(* IEC 61131-3 sources: advent-of-code/day9, 5 files *)

(* ---- demo.st ---- *)
VAR_GLOBAL CONSTANT
	rows : DINT := 5;
	cols : DINT := 10;
END_VAR

VAR_GLOBAL
	input : ARRAY[0..rows-1,0..cols -1] OF DINT :=
[
2,1,9,9,9,4,3,2,1,0,
3,9,8,7,8,9,4,9,2,1,
9,8,5,6,7,8,9,8,9,2,
8,7,6,7,8,9,6,7,8,9,
9,8,9,9,9,6,5,6,7,8
];
END_VAR

(* ---- input.st ---- *)
VAR_GLOBAL CONSTANT
	rows : DINT := 100;
	cols : DINT := 100;
END_VAR

VAR_GLOBAL
	input : ARRAY[0..rows-1,0..cols -1] OF DINT :=
[9,9,7,6,5,5,7,8,5,6,7,9,9,8,7,5,6,7,9,8,7,5,6,4,2,4,5,6,9,8,9,9,9,8,7,6,7,9,7,8,9,3,1,0,9,8,9,8,9,8,7,6,5,8,7,8,7,8,9,9,9,8,7,6,5,6,5,6,6,7,8,9,6,5,4,3,2,1,0,1,2,3,5,6,7,8,9,9,8,7,6,7,9,4,3,1,0,2,3,4,
8,7,6,5,4,3,2,1,4,5,7,8,9,9,8,3,9,8,9,8,6,4,3,2,1,3,4,5,9,7,8,9,9,9,9,5,4,5,6,9,5,3,2,9,8,7,6,7,9,9,6,5,4,2,6,5,6,7,8,9,9,8,6,5,4,2,3,4,5,7,8,9,9,6,5,4,3,2,9,4,3,9,6,9,8,9,8,7,6,6,5,6,7,9,4,4,2,5,4,5,
9,8,9,8,5,5,3,2,3,4,5,6,7,8,9,9,8,9,8,7,6,5,4,3,2,4,9,9,7,6,7,8,9,9,8,9,5,6,8,9,5,4,9,8,7,6,5,6,7,8,9,4,3,1,2,4,5,8,9,9,8,5,4,3,2,1,2,6,7,9,9,9,8,7,8,5,6,9,8,9,9,8,9,9,9,9,9,6,5,4,3,4,5,8,9,5,3,4,5,6,
8,9,8,7,6,6,8,7,6,5,6,7,9,9,9,8,7,6,9,9,8,6,7,5,3,9,8,7,6,5,6,7,9,8,7,9,9,8,9,9,6,9,8,7,6,5,4,5,6,7,8,9,1,0,1,3,4,5,6,9,7,6,5,4,3,2,3,5,6,7,8,9,9,8,9,6,7,9,7,9,8,7,8,9,9,9,8,9,5,4,2,5,5,7,8,9,4,5,9,7,
7,6,9,8,7,7,8,9,7,8,8,9,5,1,2,9,9,5,4,3,9,7,8,6,4,7,9,7,5,4,3,4,4,5,6,7,8,9,7,8,9,3,9,9,8,8,3,6,7,8,9,5,2,1,2,4,6,7,8,9,9,8,7,5,5,3,4,5,6,8,9,9,9,9,9,9,9,8,6,5,7,6,7,8,9,8,7,7,4,1,0,1,3,6,7,8,9,9,8,9,
7,5,3,9,9,8,9,9,8,9,9,4,3,2,3,9,8,6,5,2,9,8,9,8,5,6,9,8,4,3,2,1,3,4,7,9,9,6,5,4,3,2,9,8,7,6,2,3,8,9,5,4,3,2,4,5,8,8,9,2,1,9,7,6,6,4,6,8,9,9,8,8,9,9,9,8,7,6,5,4,3,5,6,9,8,7,6,5,3,2,1,2,4,5,6,9,5,6,7,8,
4,3,2,1,3,9,8,9,9,1,2,9,4,3,4,5,9,7,6,1,2,9,8,7,6,9,8,6,5,5,3,3,4,6,9,9,9,7,4,3,2,1,9,7,6,5,3,5,9,9,9,5,4,3,5,7,8,9,8,9,0,9,8,9,8,8,7,8,9,8,7,6,7,8,9,9,7,5,4,3,2,4,5,6,9,8,7,6,4,3,4,5,5,7,8,9,4,5,6,7,
9,9,3,2,3,5,7,8,9,0,9,8,9,4,9,6,9,8,7,2,3,5,9,9,9,8,9,8,7,6,4,4,5,7,8,9,8,7,5,2,1,0,2,9,7,6,9,9,8,7,8,9,7,5,6,8,9,9,7,8,9,9,9,9,9,9,9,9,7,6,5,5,6,6,8,9,8,6,5,5,4,6,8,9,4,9,8,7,6,7,8,9,6,7,9,4,2,4,5,6,
7,8,9,3,4,5,9,9,3,9,8,7,8,9,8,9,9,9,8,4,9,9,9,8,9,7,8,9,8,9,8,7,6,8,9,8,7,6,4,3,2,4,4,5,9,9,8,9,6,5,7,8,9,9,7,9,4,7,5,6,7,8,9,8,8,9,9,8,7,5,4,3,4,5,9,9,9,8,6,6,5,7,9,7,5,9,9,8,9,8,9,8,7,8,9,2,1,3,4,7,
6,8,9,9,9,7,8,9,1,9,9,6,5,5,7,8,9,9,9,9,8,7,8,7,5,6,7,8,9,9,9,9,7,8,9,9,8,7,5,4,3,9,5,6,9,9,7,8,9,4,6,8,9,9,8,9,3,3,4,5,8,9,8,7,7,9,8,6,5,4,3,2,3,6,7,8,9,9,8,7,6,8,9,7,6,8,9,9,2,9,3,9,8,9,8,4,2,5,6,8,
5,7,6,7,8,9,9,9,9,8,7,6,4,4,5,5,8,9,9,9,7,6,5,3,4,7,7,9,8,9,9,9,8,9,3,2,9,8,9,5,9,8,9,9,8,7,6,8,5,3,5,7,9,9,9,2,1,2,3,4,7,9,7,6,5,3,9,8,7,5,4,3,5,6,7,8,9,2,9,8,9,9,9,8,7,9,2,0,1,9,1,0,9,9,7,5,4,9,8,9,
4,3,5,6,8,9,9,9,8,7,6,4,3,2,3,4,7,8,9,9,8,7,4,1,3,5,6,6,7,8,9,9,9,8,9,1,2,9,8,9,8,7,9,9,8,7,5,3,1,2,3,8,9,9,4,3,0,1,6,5,6,9,8,7,6,4,5,9,8,9,5,9,6,7,8,9,4,3,4,9,2,1,0,9,8,9,3,9,9,8,9,1,9,8,7,6,9,8,9,9,
3,2,4,5,6,8,9,9,9,8,4,3,2,1,2,4,5,6,8,9,9,8,3,0,2,3,4,5,6,7,8,9,8,7,8,9,3,9,7,9,7,6,9,8,9,8,7,5,0,1,2,6,7,8,9,2,1,2,7,9,7,8,9,9,7,8,7,8,9,8,9,8,9,8,9,9,8,6,5,6,9,9,9,9,9,9,9,8,8,7,8,9,9,9,8,9,8,7,8,9,
4,3,4,6,8,9,7,9,9,8,5,4,3,3,4,5,6,8,9,8,6,3,2,1,2,5,5,8,7,8,9,7,9,6,9,9,9,8,6,8,7,5,7,7,8,9,9,4,2,3,3,4,5,9,9,4,3,3,4,5,8,9,9,8,9,9,9,9,8,7,7,7,8,9,9,9,9,7,6,9,8,7,8,9,9,9,8,7,6,5,7,8,9,9,9,8,7,6,4,5,
6,5,6,7,9,7,6,6,9,7,6,5,4,5,7,6,7,9,7,6,5,4,3,2,3,5,6,7,8,9,6,5,4,5,9,8,7,6,5,4,6,4,5,6,7,9,6,4,3,5,4,5,6,7,8,9,4,5,5,7,9,9,8,7,8,9,9,8,9,6,5,6,9,9,9,8,9,8,9,8,7,6,9,9,9,8,7,4,5,4,5,6,7,8,9,9,8,4,3,4,
7,9,8,8,9,6,5,4,9,8,8,6,5,6,8,7,8,9,9,8,7,5,4,3,4,5,7,8,9,8,7,8,5,6,9,9,8,7,6,3,2,3,8,9,9,8,7,5,9,8,5,6,7,8,9,7,5,7,8,9,9,8,7,6,7,9,8,7,6,5,3,7,8,9,8,7,8,9,8,7,6,5,6,8,9,9,6,3,2,3,4,5,6,7,8,9,4,3,2,3,
8,9,9,9,6,5,4,3,1,9,9,7,6,7,9,8,9,6,7,9,8,9,5,6,5,6,8,9,4,9,8,9,6,7,8,9,9,5,4,2,1,2,7,7,8,9,8,9,8,7,6,9,8,9,8,9,6,8,9,8,9,9,6,5,6,6,9,8,7,6,5,6,7,8,9,6,4,3,9,8,7,6,7,9,9,8,5,4,3,5,5,9,8,9,9,9,5,4,3,4,
9,4,9,8,7,6,5,4,2,3,4,9,8,8,9,9,6,5,6,7,9,8,7,7,9,8,9,4,3,2,9,8,7,8,9,9,8,7,4,3,2,3,5,6,7,8,9,9,9,8,8,9,9,6,7,8,9,9,8,7,7,6,5,4,5,5,4,9,8,7,6,7,8,9,8,9,3,2,1,9,9,7,8,9,8,7,6,9,8,6,6,7,9,8,7,8,9,6,4,5,
4,3,4,9,8,7,6,4,3,4,5,9,9,9,9,9,3,4,8,9,3,9,8,8,9,9,8,6,4,4,5,9,8,9,9,9,9,9,8,7,3,4,5,7,8,9,9,9,8,9,9,4,4,5,7,8,9,8,7,6,6,5,4,2,4,4,3,4,9,8,7,9,9,6,7,8,9,3,4,5,9,8,9,6,9,8,9,9,8,7,7,8,9,5,6,7,8,9,5,6,
3,2,5,6,9,8,7,5,9,5,9,8,9,8,8,8,9,9,9,4,2,3,9,9,4,3,9,9,5,7,8,9,9,7,8,7,9,9,9,6,5,6,8,9,9,8,9,8,7,6,5,3,2,1,6,7,8,9,6,5,4,3,2,1,0,1,2,3,4,9,8,9,6,5,7,9,9,4,9,7,8,9,3,4,5,9,9,9,9,8,9,9,2,4,5,6,9,9,6,9,
4,3,4,5,6,9,8,9,8,9,8,6,5,6,7,6,7,8,9,2,1,2,3,4,9,2,9,8,9,9,9,8,7,5,4,5,7,8,9,9,6,8,9,7,6,7,4,9,9,8,6,4,4,3,4,5,7,8,9,7,5,9,9,3,1,5,3,5,6,9,9,6,5,4,5,6,8,9,8,9,9,3,2,3,4,9,9,8,9,9,9,2,1,2,4,7,9,8,9,8,
9,5,5,9,8,9,9,8,7,6,5,4,3,1,3,4,6,9,4,3,2,5,4,9,8,9,8,7,8,9,9,7,6,4,3,4,5,6,9,8,7,9,7,6,5,4,3,9,8,7,6,5,6,7,5,6,7,8,9,9,9,7,8,9,2,3,4,6,9,8,5,4,3,2,3,4,5,6,7,8,9,4,3,9,9,8,7,7,7,8,7,9,9,3,9,9,8,7,8,7,
7,9,9,8,9,4,2,9,6,5,4,2,1,0,1,2,3,4,9,4,3,4,9,9,7,8,7,6,7,9,8,6,2,1,2,3,4,8,9,9,9,9,9,8,6,5,2,3,9,9,7,7,7,8,8,7,8,9,9,8,7,6,9,8,9,4,6,9,8,7,6,5,2,1,2,6,9,8,9,9,7,5,9,8,9,5,6,6,5,4,6,8,8,9,8,7,6,5,4,6,
6,8,9,7,8,9,1,9,7,7,6,3,2,1,6,3,7,6,8,9,4,9,8,7,6,5,6,5,6,8,9,5,4,0,1,3,5,6,7,9,9,9,8,7,5,2,1,4,5,6,9,8,8,9,9,8,9,8,7,7,6,5,8,7,7,9,9,9,9,8,7,6,3,2,3,4,9,9,1,0,9,9,8,7,7,4,5,2,3,3,5,6,7,9,9,8,5,4,3,4,
5,9,5,6,7,8,9,8,7,6,5,4,3,2,4,5,6,8,9,7,6,9,9,5,4,4,3,4,5,7,8,9,3,2,3,4,8,7,9,9,9,8,9,5,4,3,2,3,4,9,9,9,9,5,4,9,8,7,6,5,4,4,6,5,6,8,8,9,9,9,9,5,4,7,5,6,7,8,9,1,9,8,7,6,5,3,2,1,0,2,5,8,9,9,9,7,4,3,2,3,
3,3,4,7,9,7,9,9,9,7,6,5,9,4,5,6,7,8,9,8,9,8,7,4,3,1,2,5,5,6,7,8,9,6,5,5,6,9,9,9,8,7,8,9,5,6,3,9,9,8,7,6,7,4,3,4,9,8,9,4,3,3,3,4,5,6,7,8,9,9,9,7,5,6,7,8,9,9,8,9,8,9,8,7,6,4,3,2,1,3,4,6,7,9,7,6,5,4,3,4,
1,2,3,4,5,6,7,9,9,8,7,6,7,7,6,8,9,9,9,9,8,7,6,5,9,0,1,2,3,8,9,9,8,7,6,6,9,8,9,8,7,6,7,8,9,8,9,8,9,9,5,4,3,4,2,3,4,9,8,3,2,1,2,3,4,7,9,9,9,9,8,7,6,9,8,9,5,4,6,9,7,6,9,8,7,5,6,3,2,4,5,6,7,8,9,7,6,7,5,5,
3,5,6,9,6,7,8,9,6,9,8,8,9,8,7,9,8,9,8,9,9,8,7,9,8,9,2,3,5,6,8,9,9,8,7,9,8,7,8,9,6,5,9,9,9,9,9,6,9,8,9,5,2,0,1,2,9,8,7,5,3,3,3,4,5,6,7,8,9,1,9,8,7,8,9,5,4,3,9,7,6,5,9,8,7,6,7,5,6,5,6,7,8,9,9,8,8,7,6,7,
4,6,7,8,9,8,9,6,5,7,9,9,6,9,9,8,7,8,7,8,9,9,9,8,7,8,9,4,5,6,7,9,9,9,9,7,9,6,7,8,9,4,5,8,9,9,7,5,6,7,8,9,2,1,2,4,5,9,8,9,6,5,6,7,9,7,8,9,5,3,9,9,8,9,9,8,5,9,8,6,5,4,3,9,9,8,9,9,7,7,7,8,9,3,2,9,9,8,7,8,
6,9,8,9,2,9,8,7,4,3,2,3,5,9,8,7,6,5,6,7,9,9,9,8,6,7,8,9,7,8,9,3,9,8,7,6,8,5,9,9,4,3,4,6,9,8,6,4,5,6,9,8,9,2,4,5,9,9,9,8,7,7,9,8,9,8,9,7,6,9,8,6,9,8,9,7,6,9,8,7,6,5,4,7,8,9,6,7,9,8,9,9,6,5,4,5,9,9,8,9,
7,8,9,2,0,1,9,6,5,1,0,1,9,8,7,6,5,4,5,8,9,9,8,7,5,6,7,8,9,9,0,2,3,9,8,4,3,4,8,9,3,2,1,9,8,6,5,3,4,5,6,7,8,9,5,9,8,9,9,9,8,9,3,9,5,9,9,8,9,8,7,5,6,7,8,9,9,9,9,8,9,6,5,6,9,5,4,6,5,9,9,9,9,6,5,9,8,7,9,6,
8,9,8,9,1,9,8,7,7,2,1,2,4,9,8,5,4,3,4,5,9,9,9,8,9,8,8,9,7,8,9,3,4,9,6,5,2,5,7,8,9,9,9,8,9,8,4,2,3,4,9,8,9,9,9,8,7,8,9,8,9,0,1,2,3,9,9,9,9,9,6,4,6,7,9,6,8,9,9,9,9,7,6,7,8,9,3,3,4,9,8,9,8,9,6,9,7,6,5,4,
9,6,7,8,9,4,9,9,8,9,2,3,4,9,9,7,5,2,3,6,7,8,9,9,2,9,9,7,6,7,8,9,9,8,5,4,3,4,5,6,7,8,9,7,8,9,2,1,2,3,4,9,8,9,8,9,5,6,5,7,8,9,9,3,9,8,9,8,9,8,7,3,1,2,3,4,6,7,9,9,9,8,9,8,9,3,2,1,9,8,7,6,7,9,7,9,8,7,9,3,
3,5,6,8,9,3,1,0,9,8,9,4,9,8,8,6,2,1,2,7,8,9,7,5,1,0,3,4,5,6,7,9,8,7,6,5,4,5,6,7,8,9,8,6,9,8,9,0,1,2,9,8,7,9,7,5,4,3,4,9,9,9,8,9,8,7,6,7,8,9,8,2,0,1,2,4,5,6,7,8,9,9,9,9,9,9,1,0,1,9,9,5,6,8,9,9,9,9,8,9,
8,6,8,9,5,4,3,9,8,7,8,9,8,7,7,5,1,0,2,4,5,7,9,4,2,1,2,3,4,5,7,9,9,8,8,6,5,6,8,9,9,6,5,4,5,7,9,9,2,9,9,9,6,9,7,6,2,1,9,8,9,8,7,5,4,6,5,6,9,8,9,3,1,4,3,5,7,8,9,9,6,7,9,8,9,8,9,1,3,9,8,4,5,9,9,9,9,8,7,6,
8,7,9,7,6,9,9,8,7,6,9,8,7,6,5,4,3,2,3,5,6,8,9,4,3,2,3,4,5,6,7,9,8,9,9,7,6,7,9,9,9,5,4,3,5,4,9,8,9,8,7,6,5,4,3,2,1,0,1,7,8,9,5,4,3,2,4,9,8,7,8,9,2,3,8,7,9,9,1,3,4,9,8,7,7,6,8,9,9,8,7,3,7,8,9,8,9,7,6,5,
9,8,9,8,9,8,7,6,5,4,5,9,9,8,7,5,4,6,4,8,9,9,7,5,4,3,4,5,7,8,9,8,7,6,9,8,8,8,9,8,8,9,0,1,2,3,9,7,6,9,9,8,6,7,9,6,3,3,2,6,7,8,9,3,2,1,9,8,7,6,7,8,9,9,9,8,9,1,0,5,9,8,7,6,5,5,7,8,9,9,6,5,6,9,8,7,6,5,4,3,
3,9,7,9,9,9,8,9,4,3,4,5,6,9,8,7,5,9,6,7,8,9,9,6,5,9,5,6,8,9,9,9,6,5,4,9,9,9,9,7,6,8,9,3,5,9,8,9,5,6,7,9,7,9,8,5,4,5,4,5,6,7,8,9,4,3,9,7,6,5,6,7,6,7,8,9,3,2,1,6,7,9,6,5,4,3,5,6,9,8,7,6,7,9,9,8,7,6,5,4,
4,5,6,8,9,8,9,8,9,4,5,6,9,9,9,8,6,8,7,8,9,2,9,7,9,8,7,7,9,1,9,8,9,4,3,4,5,9,8,6,4,7,8,9,9,8,6,5,4,5,6,7,9,8,7,6,5,6,5,6,7,9,9,6,5,9,8,7,5,4,3,5,5,6,9,8,9,4,5,9,9,8,5,4,3,2,4,5,6,9,9,7,8,9,9,9,9,7,6,5,
5,6,9,9,8,7,6,7,9,5,6,7,8,9,6,9,7,8,8,9,2,1,9,8,9,9,8,9,1,0,9,7,8,9,4,9,9,8,9,4,3,5,1,9,8,9,7,4,3,4,5,6,7,9,8,7,6,7,6,7,8,9,8,7,9,8,7,6,4,3,2,3,4,5,6,7,8,9,9,8,7,6,5,4,2,1,2,3,4,7,9,8,9,9,9,8,7,9,7,6,
6,9,8,9,9,6,5,6,8,9,7,8,9,4,5,9,8,9,9,5,4,2,4,9,8,9,9,9,9,9,8,6,7,8,9,8,7,6,4,3,2,1,0,5,7,8,9,3,2,3,4,5,6,7,9,8,7,8,7,8,9,8,9,8,9,9,8,7,9,2,1,2,3,6,7,6,8,9,9,9,6,5,4,3,2,0,1,4,5,6,7,9,2,9,8,7,6,9,8,7,
9,9,7,6,8,6,4,5,7,8,9,9,4,3,4,4,9,8,9,6,5,6,9,8,7,9,9,9,8,7,6,5,3,4,9,8,7,6,5,4,5,9,2,4,6,9,3,2,1,2,3,6,7,8,9,9,8,9,8,9,9,7,8,9,3,2,9,9,8,9,0,1,2,3,4,5,7,8,9,9,8,7,8,4,3,1,2,3,4,5,8,9,1,2,9,6,5,6,9,8,
8,9,8,5,9,2,3,4,6,7,8,9,0,1,2,3,4,7,8,9,6,8,9,7,6,8,9,9,9,8,7,6,2,1,2,9,8,7,6,6,7,8,4,5,7,8,9,1,0,1,2,3,4,9,9,9,9,3,9,9,8,5,4,3,2,1,9,8,7,9,1,9,3,4,5,6,8,9,1,2,9,8,9,5,4,4,3,4,5,6,8,9,2,9,8,9,4,5,6,9,
7,6,5,4,3,1,2,3,5,6,9,2,1,3,5,4,5,6,7,8,9,9,8,6,5,6,7,8,9,9,8,5,4,2,3,7,9,8,7,9,8,9,7,6,9,9,3,2,1,2,3,4,5,6,8,9,3,2,9,8,7,6,5,4,5,9,8,7,6,8,9,8,9,5,6,9,9,1,0,1,2,9,8,6,5,6,7,7,6,7,9,9,9,8,6,4,3,4,5,9,
7,8,4,2,1,0,1,2,3,9,8,9,2,4,6,5,6,7,9,9,9,9,6,5,4,5,6,7,9,9,9,6,5,3,4,5,7,9,8,9,9,8,9,7,8,9,4,3,2,5,4,5,6,9,9,6,5,3,9,9,8,7,6,7,6,9,7,6,5,7,9,7,8,9,7,8,9,2,3,4,5,7,9,7,8,7,8,8,9,8,9,9,9,8,7,6,4,5,7,8,
6,5,4,3,2,1,4,3,5,6,7,8,9,5,6,8,7,9,9,9,9,8,7,3,2,3,5,6,8,9,9,7,6,4,5,6,8,9,9,7,6,7,9,8,9,6,5,4,3,7,5,6,7,8,9,9,7,9,8,9,9,8,7,9,8,9,8,7,4,4,5,6,7,8,9,9,9,4,4,7,6,7,9,8,9,8,9,9,8,9,9,8,9,9,8,6,5,7,8,9,
7,6,5,4,5,2,5,4,8,7,8,9,7,6,8,9,8,9,9,8,7,6,4,2,0,1,2,4,6,7,8,9,7,5,7,8,9,9,9,6,4,3,1,9,9,7,6,7,9,8,9,8,8,9,8,9,9,8,7,9,9,9,8,9,9,9,9,9,3,2,9,7,8,9,6,7,8,9,9,9,8,8,9,9,9,9,8,7,6,7,8,7,8,9,9,7,7,8,9,7,
8,7,7,5,6,8,6,5,9,8,9,7,9,7,9,9,9,9,8,7,6,5,4,3,1,2,8,5,7,8,9,9,9,6,7,9,9,9,8,7,5,4,9,9,8,9,9,8,9,9,8,9,9,5,7,8,9,9,6,7,8,9,9,4,5,9,8,7,6,3,7,9,9,5,4,5,9,8,8,9,9,9,1,2,9,8,7,6,5,6,7,6,9,8,9,9,8,9,5,6,
9,9,8,9,8,8,7,6,7,9,8,6,5,9,8,8,9,9,9,8,9,6,5,4,2,3,7,6,7,9,8,9,8,7,8,9,9,9,9,9,6,9,8,7,7,7,8,9,9,9,7,6,5,4,6,7,8,9,5,6,9,9,6,5,6,9,9,8,5,4,6,7,8,9,3,4,5,6,7,8,9,8,9,9,9,8,6,5,4,6,6,5,6,7,8,9,9,3,4,9,
5,6,9,8,9,9,8,9,8,9,5,3,4,5,6,7,9,9,8,9,8,7,6,6,4,5,6,7,9,8,7,6,9,9,9,8,8,9,3,1,9,8,7,6,5,6,7,8,9,9,8,8,7,2,3,4,9,9,4,3,9,8,7,6,9,8,9,9,6,5,7,9,9,1,2,3,6,9,8,9,8,7,6,8,9,6,5,4,3,1,5,4,5,6,7,9,1,2,9,8,
4,5,6,7,8,9,9,9,9,8,6,7,6,9,7,9,8,8,7,6,9,9,7,7,5,6,7,9,9,9,9,5,3,2,1,6,7,8,9,9,8,9,4,3,4,5,6,7,8,9,9,9,8,3,4,5,6,8,9,2,1,9,8,9,8,7,9,8,7,6,8,9,3,2,4,4,5,6,9,7,5,4,5,9,8,7,6,5,4,0,2,3,6,7,8,9,3,9,8,7,
5,9,8,9,9,8,9,7,6,9,9,8,9,8,9,7,6,5,4,5,4,5,9,8,6,7,9,9,8,9,8,9,5,4,3,5,8,9,9,8,7,6,5,4,5,6,7,8,9,3,2,1,9,4,6,7,8,9,9,1,0,1,9,8,7,6,5,9,8,7,8,9,4,9,9,7,6,8,9,6,4,3,4,5,9,8,9,7,5,1,4,5,8,9,9,9,9,9,9,6,
6,7,9,5,6,7,8,9,9,9,9,9,8,7,9,6,5,4,3,2,3,5,6,9,7,9,9,8,7,6,7,8,9,5,4,6,9,9,9,9,8,7,6,5,6,7,8,9,8,9,4,3,4,9,7,8,9,9,8,9,1,9,8,7,6,5,4,5,9,8,9,9,9,8,8,9,7,8,9,6,5,2,6,6,7,9,5,9,7,7,6,6,8,9,8,9,8,9,8,7,
7,8,9,4,5,6,9,8,7,8,9,9,7,6,8,9,6,3,2,1,2,3,9,9,8,9,8,9,6,5,6,9,7,6,9,7,9,9,8,1,9,8,7,6,9,8,9,6,7,9,6,4,5,9,8,9,9,8,7,8,9,9,9,9,7,4,3,4,5,9,9,8,7,6,7,9,9,9,7,5,4,3,4,8,9,5,4,2,9,8,7,8,9,6,7,9,7,6,9,9,
8,9,3,2,3,9,8,7,6,7,5,8,6,5,7,9,7,4,3,4,3,4,8,9,9,9,7,8,9,4,5,8,9,7,8,9,8,8,7,0,1,9,8,7,9,9,4,5,9,8,9,5,7,9,9,8,7,8,6,8,9,9,9,8,4,3,2,3,6,9,8,7,6,5,6,8,8,9,8,7,6,4,6,7,8,9,3,1,0,9,9,9,4,5,6,8,9,4,3,1,
9,5,4,3,9,8,7,6,5,6,3,2,3,4,8,9,8,5,4,5,7,5,6,9,8,6,5,6,9,3,4,7,8,9,9,8,7,6,5,3,2,3,9,9,1,2,3,4,9,7,8,9,9,8,7,9,6,4,5,6,7,8,9,6,5,4,3,4,9,8,9,6,7,4,5,6,7,8,9,8,9,8,7,9,9,9,9,2,9,9,8,7,5,6,7,9,7,2,1,0,
8,6,6,5,7,9,6,5,4,6,2,1,2,3,4,9,9,6,5,6,8,9,9,8,7,5,4,5,8,9,5,6,7,8,9,9,9,7,9,5,3,5,6,7,9,9,4,9,8,6,7,8,9,8,6,5,4,3,4,5,6,9,8,9,6,5,4,9,8,7,6,5,2,3,4,5,8,9,1,9,4,9,8,9,8,7,8,9,8,9,9,8,9,8,9,6,5,4,2,3,
9,9,7,6,9,8,7,6,3,2,1,0,1,4,6,7,8,9,6,7,9,8,5,5,4,4,3,6,7,8,9,7,8,9,4,3,9,8,9,6,9,8,7,8,9,8,9,8,7,5,6,7,9,6,5,4,3,2,3,4,5,6,7,8,9,6,9,8,8,7,4,3,1,3,3,7,9,9,0,1,3,4,9,8,7,6,7,8,7,8,9,9,6,9,8,7,6,6,7,5,
5,6,9,8,9,9,9,5,4,3,2,3,2,3,4,5,6,9,7,9,8,7,4,3,2,1,2,4,5,9,2,9,9,5,4,2,3,9,9,7,9,9,9,9,6,7,8,9,6,4,5,9,8,7,6,5,2,1,2,5,6,8,9,9,9,9,8,7,7,6,2,1,0,1,2,6,7,8,9,9,9,9,8,7,6,5,9,8,6,8,9,7,5,6,9,8,9,7,7,6,
3,5,6,9,8,9,8,6,7,4,3,4,6,5,5,6,7,8,9,9,9,6,5,4,9,0,3,6,6,9,3,9,8,7,5,4,9,9,7,9,3,2,3,4,5,6,7,8,9,3,4,5,9,8,7,4,3,2,7,6,8,9,9,9,9,8,7,6,5,4,3,2,1,2,3,4,5,9,8,7,8,9,9,8,9,4,3,4,5,6,8,9,3,4,5,9,5,9,8,7,
8,6,9,8,7,9,8,7,6,5,4,5,6,6,8,7,8,9,9,9,8,9,6,9,8,9,4,5,7,8,9,9,9,9,7,9,8,7,6,5,4,4,4,5,7,8,9,9,3,2,3,4,8,9,6,5,4,5,6,7,9,9,8,8,7,9,8,7,6,5,4,3,8,7,5,6,7,8,9,5,7,8,9,9,8,6,2,3,4,5,7,8,9,9,6,9,4,5,9,8,
9,9,8,7,6,5,9,8,7,8,7,6,7,7,9,8,9,9,9,8,7,8,9,8,7,9,5,7,8,9,7,8,8,9,9,9,9,8,7,9,5,5,6,9,8,9,6,5,4,3,4,6,7,9,8,9,5,9,8,9,9,9,7,6,5,4,9,8,8,7,6,5,9,8,6,7,8,9,5,4,8,9,8,7,6,5,3,4,6,6,9,9,9,8,9,8,9,9,9,9,
5,6,9,9,8,4,5,9,8,9,9,7,9,8,9,9,2,9,8,7,6,7,8,9,6,8,9,8,9,8,6,5,7,8,9,9,8,9,8,9,6,6,9,9,9,8,7,6,5,4,5,7,8,9,9,7,6,7,9,9,9,8,9,5,3,2,6,9,9,8,7,6,7,9,9,8,9,6,5,3,4,5,9,9,7,6,4,5,9,7,8,9,8,7,7,6,7,8,9,9,
4,9,8,7,6,3,1,2,9,6,9,8,9,9,3,2,1,0,9,6,5,6,3,5,5,7,8,9,9,7,5,4,6,7,9,8,7,8,9,8,7,9,8,8,8,9,9,7,6,7,6,9,9,7,9,9,7,8,9,9,8,7,8,9,4,3,5,6,7,9,8,7,8,9,9,9,8,7,9,4,6,9,9,9,8,7,5,6,7,8,9,8,9,6,6,4,6,7,8,9,
3,9,8,6,5,4,2,3,4,5,6,9,8,6,5,4,9,9,8,7,4,3,2,3,4,6,7,8,9,5,4,3,8,9,8,7,6,5,6,9,8,9,7,6,7,9,8,9,9,8,7,8,9,6,7,9,8,9,8,7,7,6,9,8,9,4,5,7,9,7,9,8,9,9,9,9,9,9,8,9,9,8,9,9,9,8,6,7,8,9,8,7,6,5,4,3,4,8,9,0,
4,9,8,7,6,5,3,4,5,7,7,8,9,7,9,9,7,7,5,8,1,0,1,2,4,5,8,9,6,4,3,2,9,8,7,6,5,4,5,6,9,8,6,5,6,5,6,7,8,9,8,9,5,5,6,2,9,9,9,5,6,5,6,7,8,9,6,8,9,6,5,9,9,8,7,8,9,8,7,8,8,7,8,9,9,9,9,8,9,2,9,8,5,4,3,2,4,6,9,1,
5,6,9,8,7,6,7,8,7,8,8,9,2,9,8,7,6,5,4,3,2,1,2,3,8,8,9,9,9,5,5,1,2,9,8,9,2,3,4,9,8,7,6,4,6,4,8,9,9,9,9,5,4,3,2,1,9,8,8,4,3,4,7,7,8,9,7,9,9,9,3,2,3,4,5,9,7,6,5,6,7,6,9,9,8,7,9,9,0,1,3,9,9,2,0,1,3,9,8,9,
9,9,7,9,8,7,8,9,8,9,9,9,1,0,9,8,7,7,5,5,4,3,6,4,6,7,8,9,8,7,6,3,9,9,9,8,9,4,9,8,7,6,5,3,4,3,4,8,7,8,9,6,5,4,6,2,9,7,6,5,2,3,4,6,9,6,9,7,8,8,9,1,2,3,9,9,8,3,4,3,4,5,8,9,9,6,9,5,3,2,4,9,8,9,3,2,9,9,7,8,
8,7,6,7,9,8,9,7,9,6,7,8,9,9,8,9,9,8,7,6,5,5,7,5,7,8,9,9,9,8,7,9,8,8,6,7,8,9,9,7,6,5,4,2,1,2,3,4,6,7,9,7,7,5,7,9,8,6,5,4,3,4,5,7,9,5,6,5,6,7,8,9,3,9,8,7,3,2,1,2,5,6,7,8,9,5,8,9,4,3,9,8,7,8,9,9,8,9,6,7,
7,6,5,6,8,9,6,5,4,5,6,7,8,9,7,6,5,9,8,8,6,6,8,6,9,9,9,8,9,9,9,8,7,6,5,1,2,9,8,7,6,5,4,3,0,1,2,3,7,8,9,8,8,6,8,9,9,7,6,5,4,5,7,9,5,4,4,4,5,6,7,8,9,8,7,5,4,5,2,3,8,7,8,9,3,4,7,8,9,9,8,7,6,7,9,8,7,6,5,6,
9,7,3,8,9,9,8,4,3,7,8,9,9,8,6,5,3,2,9,8,7,7,9,7,8,9,5,6,7,9,8,7,6,5,4,3,3,4,9,6,5,4,3,2,1,2,5,7,8,9,9,9,9,7,8,9,9,8,7,8,5,9,8,9,4,3,2,3,4,5,6,7,8,9,8,6,5,6,3,5,9,8,9,5,4,5,6,7,9,6,9,6,5,9,8,7,6,5,4,4,
7,6,2,9,6,8,9,5,4,5,6,7,8,9,7,4,3,1,0,9,8,9,9,8,9,4,3,2,3,4,9,9,8,6,5,9,5,9,8,7,8,5,4,3,2,3,4,5,6,8,9,3,9,8,9,1,2,9,8,9,6,7,9,2,1,0,1,5,6,7,8,9,9,9,9,7,6,5,4,5,6,9,7,6,7,6,7,9,8,5,4,5,4,6,9,8,5,4,3,3,
5,4,3,4,5,7,8,9,5,9,8,9,9,7,6,5,4,5,1,3,9,8,9,9,6,5,4,5,6,8,9,5,9,7,6,8,9,8,9,8,9,6,5,4,5,4,5,7,8,9,1,2,4,9,4,2,9,8,9,8,7,8,9,3,2,4,3,4,5,9,9,9,8,9,9,9,8,6,7,6,8,9,9,7,8,8,9,8,7,6,3,4,3,4,5,9,9,2,1,2,
6,5,4,5,7,8,9,7,6,7,9,5,3,9,8,6,5,3,2,5,6,7,9,8,7,8,5,6,7,8,9,4,9,8,7,9,8,7,6,9,9,7,6,5,7,9,7,8,9,8,9,4,9,9,9,9,8,7,9,9,8,9,5,4,9,5,6,5,9,8,7,8,7,8,9,5,9,7,9,7,9,9,9,8,9,9,8,7,6,6,2,1,2,5,9,8,8,3,0,1,
7,8,5,6,8,9,2,9,7,9,8,9,2,3,9,7,6,4,5,6,9,8,9,9,8,9,6,9,8,9,2,3,5,9,9,8,9,6,5,6,7,9,7,6,7,9,8,9,6,7,9,9,8,9,8,9,7,6,5,6,9,8,7,9,8,9,7,9,8,7,6,7,6,7,9,6,9,8,9,9,9,9,6,9,9,8,7,6,5,4,3,0,1,9,8,7,6,3,1,2,
8,7,6,9,9,2,1,9,8,9,7,9,9,4,9,8,7,7,6,7,8,9,5,6,9,8,7,8,9,9,9,4,5,9,8,7,6,5,4,5,7,9,8,7,8,9,9,4,5,6,9,8,7,8,7,8,9,5,4,5,6,9,9,9,7,6,9,8,7,6,5,8,5,6,8,9,9,9,9,9,9,8,5,6,7,9,8,7,6,5,3,2,3,6,9,9,5,4,2,3,
9,8,7,8,9,3,2,9,9,8,6,8,8,9,9,9,9,8,7,8,9,3,4,9,9,9,8,9,6,9,8,9,9,8,7,6,5,4,3,4,9,8,9,8,9,0,1,9,9,9,8,7,6,5,6,9,6,5,3,4,5,9,8,7,6,5,6,9,8,7,4,3,4,5,6,7,8,9,9,8,7,6,4,3,9,7,9,8,7,6,5,3,4,5,9,8,6,5,6,4,
8,9,8,9,5,4,9,8,7,6,5,6,7,8,9,6,8,9,8,9,9,2,9,8,9,7,9,6,5,8,7,8,9,9,9,8,7,3,2,5,6,7,9,9,3,1,9,8,7,6,5,4,5,4,5,8,9,3,2,3,9,8,7,6,5,4,5,9,8,7,3,2,3,4,8,9,9,1,0,9,8,7,6,4,9,6,4,9,9,7,6,4,5,6,7,9,8,7,7,5,
7,4,9,7,6,5,7,9,8,8,4,5,6,9,5,4,5,5,9,7,8,9,8,7,6,5,7,2,4,5,6,7,9,9,8,7,5,4,5,6,7,8,9,8,9,9,9,9,6,5,4,3,2,3,6,7,8,9,1,2,9,7,6,6,4,3,4,5,9,6,5,4,4,5,9,5,4,3,9,9,9,8,7,9,8,4,3,2,9,8,9,9,8,7,8,9,9,8,8,9,
6,5,6,9,8,7,8,9,9,9,5,6,7,8,9,3,2,4,5,6,9,9,7,9,8,3,4,1,2,4,8,6,7,8,9,9,9,5,7,8,9,9,8,6,5,8,7,8,9,6,5,4,1,2,7,6,7,9,2,9,7,6,5,4,3,2,3,9,8,7,9,6,5,6,8,9,5,9,8,9,9,9,8,9,7,5,2,1,2,9,9,9,9,9,9,9,8,9,9,6,
7,6,9,8,9,8,9,9,9,8,6,8,8,9,3,2,1,3,4,9,8,7,6,5,3,2,1,0,2,3,4,5,6,9,8,7,8,9,8,9,8,7,6,5,4,5,6,9,9,9,4,3,2,3,4,5,6,8,9,7,9,8,6,5,4,3,4,8,9,9,8,7,8,7,9,9,9,8,7,8,9,9,9,9,5,4,3,9,9,8,8,9,1,3,9,8,7,8,9,5,
9,9,8,7,6,9,9,8,8,9,7,9,9,5,4,1,0,3,5,6,9,9,6,5,4,3,2,1,2,3,4,6,9,8,7,6,7,9,9,9,9,8,5,4,3,5,5,6,7,8,9,9,5,4,5,6,7,8,9,5,6,9,7,6,6,4,5,7,8,9,9,8,9,8,9,9,8,7,6,7,8,9,9,8,7,5,9,8,8,7,7,8,9,4,9,9,6,6,5,4,
9,8,7,6,5,9,7,6,7,9,8,9,9,4,3,2,1,2,3,4,9,8,7,6,5,4,5,2,3,4,5,9,8,7,6,5,6,8,9,9,8,7,6,4,2,3,4,5,6,9,9,8,7,5,7,7,8,9,3,4,9,7,9,8,7,5,6,8,9,2,1,9,3,9,9,8,7,6,5,6,7,9,3,9,8,6,9,7,6,5,6,9,9,9,8,7,5,4,4,3,
3,9,8,7,9,8,6,5,4,6,9,9,8,5,4,3,2,3,4,6,7,9,8,7,6,7,4,3,4,5,6,7,9,7,6,4,5,7,9,9,9,8,9,9,1,0,2,8,7,8,9,9,7,6,8,9,9,6,2,9,8,6,5,9,9,7,7,8,9,1,0,1,2,9,8,9,3,2,4,5,8,9,2,1,9,9,8,7,6,4,7,8,9,9,9,5,4,3,2,1,
2,1,9,9,9,7,7,6,3,4,9,8,7,6,5,7,8,4,5,7,8,9,9,9,8,7,5,4,5,6,7,9,8,8,5,3,4,6,7,8,9,9,9,8,9,1,2,3,5,9,8,9,8,7,9,7,6,5,4,9,8,8,4,3,2,9,8,9,3,2,2,2,9,8,7,6,4,3,4,6,9,5,4,5,6,8,9,8,7,2,9,9,9,9,7,6,5,2,1,0,
3,3,9,8,9,6,5,4,2,0,1,9,9,7,8,9,6,5,7,8,9,3,1,9,8,7,6,6,6,7,8,9,7,6,3,2,3,4,5,9,9,9,8,7,8,9,3,4,5,6,7,8,9,8,9,8,7,9,9,8,7,6,5,4,1,2,9,6,4,6,5,4,7,9,8,6,5,6,5,7,8,9,6,6,7,9,9,9,8,3,5,7,9,8,7,5,4,3,2,1,
9,9,8,7,8,9,6,5,5,4,2,3,9,8,9,8,7,6,8,9,9,9,0,1,9,8,9,7,7,8,9,8,7,5,2,1,2,3,4,5,9,8,7,6,9,8,9,6,9,7,9,9,5,9,6,9,9,7,6,9,8,8,6,5,4,3,9,8,9,7,6,5,6,7,9,8,7,7,9,8,9,9,9,8,9,9,8,9,5,4,5,6,7,9,8,6,5,4,3,2,
8,7,6,6,7,9,9,6,6,9,9,9,9,9,2,9,8,7,9,1,9,8,9,9,8,9,9,8,8,9,8,9,8,4,3,0,3,4,5,9,8,7,6,5,6,7,9,9,8,9,9,9,4,3,5,9,8,9,5,3,9,9,7,6,5,4,5,9,9,8,7,6,7,8,9,9,8,8,9,9,9,9,9,9,8,9,7,8,9,5,7,9,9,9,8,7,7,5,4,5,
9,9,5,4,6,7,8,9,9,8,7,8,9,0,1,2,9,8,9,2,9,7,8,9,7,5,4,9,9,5,7,8,9,5,2,1,2,5,6,9,8,6,5,4,5,6,8,9,7,6,7,8,9,4,9,8,7,8,9,2,0,9,8,7,6,7,6,9,9,9,8,7,8,9,4,2,9,9,9,9,8,7,9,8,7,5,6,9,9,9,8,9,1,0,9,8,7,6,9,6,
8,7,6,5,7,8,9,6,5,4,6,9,9,1,2,3,4,9,9,9,8,6,7,8,9,3,2,1,2,4,5,9,8,7,8,2,3,4,9,8,7,5,4,3,4,9,9,7,6,5,7,7,8,9,8,7,6,9,8,9,1,3,9,8,9,8,7,8,9,8,9,8,9,6,5,6,7,8,9,8,7,6,6,4,3,4,6,8,9,9,9,6,9,9,9,9,8,9,8,9,
9,9,8,6,8,9,8,9,4,3,4,8,8,9,3,9,6,9,8,7,6,5,6,9,8,9,3,2,3,5,9,8,7,6,4,3,7,9,8,7,6,5,3,2,9,8,7,6,5,4,5,6,7,8,9,6,5,5,7,8,9,4,5,9,5,9,8,9,7,6,4,9,9,8,6,7,8,9,8,7,6,5,4,3,2,1,2,7,8,9,6,5,8,7,8,9,9,8,7,8,
9,9,9,8,9,5,6,7,3,2,3,6,7,8,9,8,9,9,8,9,8,3,5,6,7,8,9,3,4,6,7,9,8,7,5,4,5,6,9,8,7,3,2,1,2,9,9,5,4,3,9,8,9,9,8,7,4,4,5,6,8,9,6,9,3,2,9,9,9,5,3,5,4,9,7,8,9,9,9,8,6,5,3,2,1,0,5,6,7,8,9,4,5,6,7,9,8,7,6,9,
9,8,9,9,5,4,2,1,0,1,4,5,6,9,9,7,9,9,7,5,4,2,4,5,6,7,8,9,5,7,9,9,9,8,9,5,7,7,8,9,8,2,1,0,1,9,8,9,4,2,8,9,9,8,7,6,2,3,4,5,8,9,7,8,9,1,0,9,8,9,2,1,2,9,8,9,8,9,9,9,7,6,4,3,5,1,4,5,6,9,9,2,1,2,9,7,7,5,5,6,
8,7,8,9,6,5,3,2,1,2,5,6,8,9,7,6,9,8,7,6,3,1,3,4,5,9,9,7,6,9,8,9,9,9,9,9,8,9,9,7,9,3,2,1,9,8,7,4,3,1,6,8,9,7,6,5,4,5,6,6,7,8,9,9,9,9,9,8,7,8,9,0,1,2,9,6,7,8,9,9,9,7,5,4,3,2,3,4,5,7,8,9,0,9,8,6,5,4,4,5,
7,6,9,8,7,6,5,3,3,3,4,5,7,8,9,5,7,9,8,5,4,5,4,5,6,7,8,9,9,9,7,8,9,9,8,9,9,8,7,6,5,4,4,9,8,7,6,5,4,3,4,7,8,9,7,9,9,6,7,7,8,9,2,1,9,8,7,7,6,7,8,9,2,3,4,5,7,8,9,8,9,8,6,5,4,3,5,7,6,7,8,9,9,8,7,5,4,3,2,3,
6,5,4,9,8,9,6,5,4,4,6,7,9,9,3,4,6,7,9,6,5,6,7,6,8,9,9,9,8,7,6,5,8,5,7,9,9,9,8,7,8,6,5,6,9,9,7,6,5,7,5,6,7,8,9,8,8,9,8,8,9,8,9,9,8,7,6,6,4,5,7,8,9,5,5,6,7,9,8,7,9,8,7,6,5,4,6,8,9,9,9,6,9,8,7,6,8,2,1,0,
5,4,3,1,9,8,7,7,5,8,9,8,9,1,2,4,5,6,9,8,6,7,9,8,9,7,9,9,9,7,5,4,6,4,6,8,9,9,9,9,9,7,6,8,9,9,8,7,9,8,6,7,8,9,5,6,7,8,9,9,6,7,9,9,8,6,5,4,3,4,6,7,8,9,6,7,9,8,7,6,7,9,9,8,7,6,8,9,9,9,6,5,6,9,9,8,9,4,3,2,
3,2,1,0,1,9,8,7,6,7,8,9,1,0,1,2,6,7,9,8,7,8,9,9,5,6,8,9,8,6,4,3,4,3,4,5,7,9,9,8,9,8,7,9,8,7,9,8,9,8,7,9,9,2,4,8,9,9,3,4,5,6,7,9,8,7,6,6,5,6,9,8,9,9,7,9,8,9,7,5,6,5,6,9,9,9,9,8,9,8,9,4,3,2,3,9,9,5,5,3,
4,5,2,3,4,5,9,8,9,8,9,4,2,1,2,3,7,8,9,9,8,9,9,8,7,8,9,7,6,5,3,2,1,2,3,4,6,8,9,7,5,9,8,9,9,5,4,9,8,9,8,9,2,1,5,6,7,9,2,3,4,5,7,8,9,8,8,7,6,7,9,9,3,2,9,8,7,6,9,4,3,4,5,6,9,8,7,6,5,7,8,9,4,1,4,9,8,7,6,4,
6,7,3,5,5,6,8,9,9,9,6,4,3,4,4,5,6,7,8,9,9,0,1,9,8,9,8,7,5,4,3,2,0,3,5,6,7,9,6,5,4,3,9,8,7,5,3,5,7,8,9,4,3,2,6,7,8,9,1,4,6,6,7,8,9,9,9,8,7,9,7,5,4,5,7,9,8,5,4,3,2,5,6,7,8,9,9,8,4,5,9,6,5,3,4,5,9,8,9,5];
END_VAR

(* ---- sol.st ---- *)
//defined elsewere rows,cols,input
FUNCTION main : DINT
VAR_TEMP
	i,j,current, count,sum : DINT := 0;
	result : ARRAY[0..rows-1,0..cols-1] OF BOOL;
	basins : list;
	basin : Point;
END_VAR

FOR i:= 0 TO rows - 1 DO
	FOR j := 0 TO cols -1 DO
		(*If value is a 9 just skip it there is nothing bigger*)
		current := input[i,j];
		IF current < 9 THEN
			result[i,j] := TRUE;
			(* check up (i -1) *)
			IF i - 1 >= 0 THEN
				IF current >= input[i-1,j] THEN
					result[i,j] := FALSE;
				END_IF
			END_IF
			(* check down (i + 1) *)
			IF i + 1 < rows THEN
				IF current >= input[i+1,j] THEN
					result[i,j] := FALSE;
				END_IF
			END_IF
			(* check up (j -1) *)
			IF j - 1 >= 0 THEN
				IF current >= input[i,j-1] THEN
					result[i,j] := FALSE;
				END_IF
			END_IF
			(* check down (j + 1) *)
			IF j + 1 < cols THEN
				IF current >= input[i,j+1] THEN
					result[i,j] := FALSE;
				END_IF
			END_IF
		ELSE
			result[i,j] := FALSE;
		END_IF
	END_FOR
END_FOR

FOR i:= 0 TO rows - 1 DO
	FOR j := 0 TO cols -1 DO
		IF result[i,j] THEN
			count := count + 1;
			sum := sum + input[i,j] + 1;
			basin.y := i;
			basin.x := j;
			basins.add(calc_basin_size(&input,basin));
		END_IF
	END_FOR
END_FOR

printf('Count %d, Sum %d $n', count, sum);
printf('Basins %d,%d,%d, * %d$n', basins.get(0), basins.get(1), basins.get(2), basins.get(0) * basins.get(1) * basins.get(2));

END_FUNCTION

FUNCTION calc_basin_size : DINT
VAR_INPUT
	grid : REF_TO ARRAY[0..rows-1, 0..cols-1] OF DINT;
	basin_start : Point;
END_VAR
VAR_TEMP
	candidates : Stack;
	current : Point;
	pt : Point;
	visited : ARRAY[0..rows-1, 0..cols-1] OF BOOL := [10000(FALSE)];
	size : DINT := 0;
END_VAR
	candidates.push(basin_start);

	WHILE NOT candidates.is_empty() DO
		size := size + 1;
		current := candidates.pop();
		visited[current.y,current.x] := TRUE;
		(* check up (i -1) *)
		IF (current.y - 1) >= 0 THEN
			pt.x := current.x;
			pt.y := current.y - 1;
			IF grid^[pt.y,pt.x] < 9 AND NOT visited[pt.y,pt.x] THEN
				candidates.push(pt);
			END_IF
			visited[pt.y,pt.x] := TRUE;
		END_IF
		(* check down (i + 1) *)
		IF (current.y + 1) < rows THEN
			pt.x := current.x;
			pt.y := current.y + 1;
			IF grid^[pt.y,pt.x] < 9 AND NOT visited[pt.y,pt.x] THEN
				candidates.push(pt);
			END_IF
			visited[pt.y,pt.x] := TRUE;
		END_IF
		(* check up (j -1) *)
		IF (current.x - 1) >= 0 THEN
			pt.x := current.x - 1;
			pt.y := current.y;
			IF grid^[pt.y,pt.x] < 9 AND NOT visited[pt.y,pt.x] THEN
				candidates.push(pt);
			END_IF
			visited[pt.y,pt.x] := TRUE;
		END_IF
		(* check down (j + 1) *)
		IF (current.x + 1) < cols THEN
			pt.x := current.x + 1;
			pt.y := current.y;
			IF grid^[pt.y,pt.x] < 9 AND NOT visited[pt.y,pt.x] THEN
				candidates.push(pt);
			END_IF
			visited[pt.y,pt.x] := TRUE;
		END_IF
	END_WHILE

	calc_basin_size := size;
	printf('%d$n', size);

END_FUNCTION

(* ---- list.st ---- *)
(* A list that only keeps the biggest elements *)
CLASS list
VAR
	arr : ARRAY[0..2] OF DINT;
	lowestIdx : DINT := 0;
END_VAR

METHOD add : __VOID
VAR_INPUT
	val : DINT;
END_VAR
VAR_TEMP
	i, lowest : DINT := 0;
END_VAR

IF arr[lowestIdx] < val THEN
	arr[lowestIdx] := val;

	FOR i := 0 TO 2 DO
		IF arr[i] < arr[lowest] THEN
			lowest := i;
		END_IF
	END_FOR

	lowestIdx := lowest;
END_IF

END_METHOD

METHOD get : DINT
VAR_INPUT loc : DINT; END_VAR
	get := arr[loc];
END_METHOD

END_CLASS

(* ---- stack.st ---- *)
CLASS Stack
VAR
	arr : ARRAY[0..cols*rows] OF Point;
	counter : DINT := 0;
END_VAR

METHOD push : __VOID
	VAR_INPUT
		p : Point;
	END_VAR
	arr[counter] := p;
	counter := counter + 1;
END_METHOD

METHOD pop : Point
	counter := counter - 1;
	IF counter < 0 THEN
		counter := 0;
	END_IF
	pop := arr[counter];
END_METHOD

METHOD peek : Point
	peek := arr[counter - 1];
END_METHOD

METHOD is_empty : BOOL
	is_empty := counter = 0;
END_METHOD

END_CLASS
